FUNCTION_BLOCK MC2_Axis_Base EXTENDS CyclicBase
VAR_INPUT
END_VAR
VAR_OUTPUT
END_VAR
VAR
	_axis : Tc2_MC2.AXIS_REF;
	axesEnable		: AxisPower(_axis);
	axesResetCommand		: AxesReset(_axis);
	axesMoveToCommand 		: Mc2MoveToPosition(_axis);
	axesHaltCommand 		: Mc2Halt(_axis);
	axesReadError : Tc2_MC2.MC_ReadAxisError;
	_MoverErrorId: DWORD;
END_VAR

{analysis -2}

METHOD Cycle : HRESULT
VAR_INPUT
END_VAR
Cycle := axesMoveToCommand.Cycle();
Cycle := axesHaltCommand.Cycle();
Cycle := axesResetCommand.Cycle();
_axis.ReadStatus();
Cycle := axesEnable.Cycle();
axesReadError(Axis := _axis, Enable := TRUE, AxisErrorID => _MoverErrorId);
END_METHOD

METHOD PUBLIC DisableAxis : BOOL
VAR_INPUT
END_VAR
DisableAxis := axesEnable.Disable();
END_METHOD

METHOD PUBLIC EnableAxis : BOOL
VAR_INPUT
END_VAR
EnableAxis := axesEnable.Enable();
END_METHOD

METHOD PUBLIC HaltAxis : BOOL
VAR
	haltResult : BOOL;
	abortResult : BOOL;
END_VAR
IF NOT axesHaltCommand.Busy THEN
	haltResult := axesHaltCommand.Execute();
	abortResult := axesMoveToCommand.Abort();
	HaltAxis := haltResult AND abortResult;
ELSE 
	HaltAxis := FALSE;
END_IF
END_METHOD

METHOD hasError : BOOL
VAR_INPUT
END_VAR
hasError := _axis.Status.Error;
END_METHOD

METHOD isAtPosition : BOOL
VAR_INPUT
	position : MC_LREAL;
END_VAR
IF _axis.NcToPlc.ActPos < position + 0.2 AND _axis.NcToPlc.ActPos > position - 0.2 THEN
	isAtPosition := TRUE;
ELSE
	isAtPosition := FALSE;
END_IF
END_METHOD

METHOD isEnabled : BOOL
VAR_INPUT
END_VAR
isEnabled := not _axis.Status.Disabled;
END_METHOD

METHOD PUBLIC isStationary : BOOL
VAR_INPUT
END_VAR
isStationary := _axis.NcToPlc.SetVelo = 0;
END_METHOD

METHOD PUBLIC MoveToPosition : BOOL
VAR_INPUT
	Position : MC_LREAL;
	Velocity : MC_LREAL;
END_VAR
IF NOT isAtPosition(position := Position) THEN
	IF NOT axesMoveToCommand.Busy THEN
		axesMoveToCommand.MoveTo(Position := Position, Velocity := Velocity);
		MoveToPosition := TRUE;
	END_IF
ELSE
	MoveToPosition := FALSE;
END_IF
END_METHOD

METHOD PUBLIC ResetAxis : BOOL
VAR
	ResetResult : BOOL;
	MoveAbortResult : BOOL;
	HaltAbortResult : BOOL;
END_VAR
ResetResult := axesResetCommand.Execute();
MoveAbortResult := axesMoveToCommand.Abort();
HaltAbortResult := axesHaltCommand.Abort();
ResetAxis := ResetResult AND MoveAbortResult AND HaltAbortResult;
END_METHOD

END_FUNCTION_BLOCK

(* stored: Version 1.1.0.1, ProductVersion 3.1.4024.12
   POU MC2_Axis_Base: Id {6091fbf5-8563-4c3d-a46f-a871d52562e9}, SpecialFunc None
   Method Cycle: Id {6e2b69ab-f1bf-4962-bdbb-f480f753daf6}
   Method DisableAxis: Id {4ca2c35a-d664-47dd-b699-e212d5be22eb}
   Method EnableAxis: Id {a835c18f-6175-4614-a6ac-65491f5fc70d}
   Method HaltAxis: Id {b5b4d676-a559-4d25-8571-0c2ec9c3c015}
   Method hasError: Id {ca345aeb-702e-4d9d-ada0-0eb76d61a85d}
   Method isAtPosition: Id {a3fbba8b-aebd-4df9-9a9b-10d926ce7c0a}
   Method isEnabled: Id {460678ae-c472-4e27-a376-f3d29d1278b6}
   Method isStationary: Id {4df49a98-73c3-4028-9049-ecd2a431e2f1}
   Method MoveToPosition: Id {bca42834-4b90-4808-be50-ee67839e4111}
   Method ResetAxis: Id {bd5b60f2-6a45-4850-931f-c2efbdee4a44} *)
